FUNCTION_BLOCK F_LEN (* string length function *)
  (* Standard: 61131-3; Classification: standard function of character string *)
  (* Version 0.0, 2013-04-25, 4DIAC-IDE, 4DIAC-Consortium *)
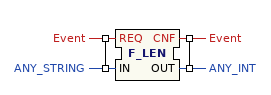
  EVENT_INPUT
    REQ WITH IN; (* Service Request *)
  END_EVENT
  EVENT_OUTPUT
    CNF WITH OUT; (* Confirmation of Requested Service *)
  END_EVENT
  VAR_INPUT
    IN : ANY_STRING; (* input string *)
  END_VAR
  VAR_OUTPUT
    OUT : ANY_INT; (* length *)
  END_VAR
END_FUNCTION_BLOCK
